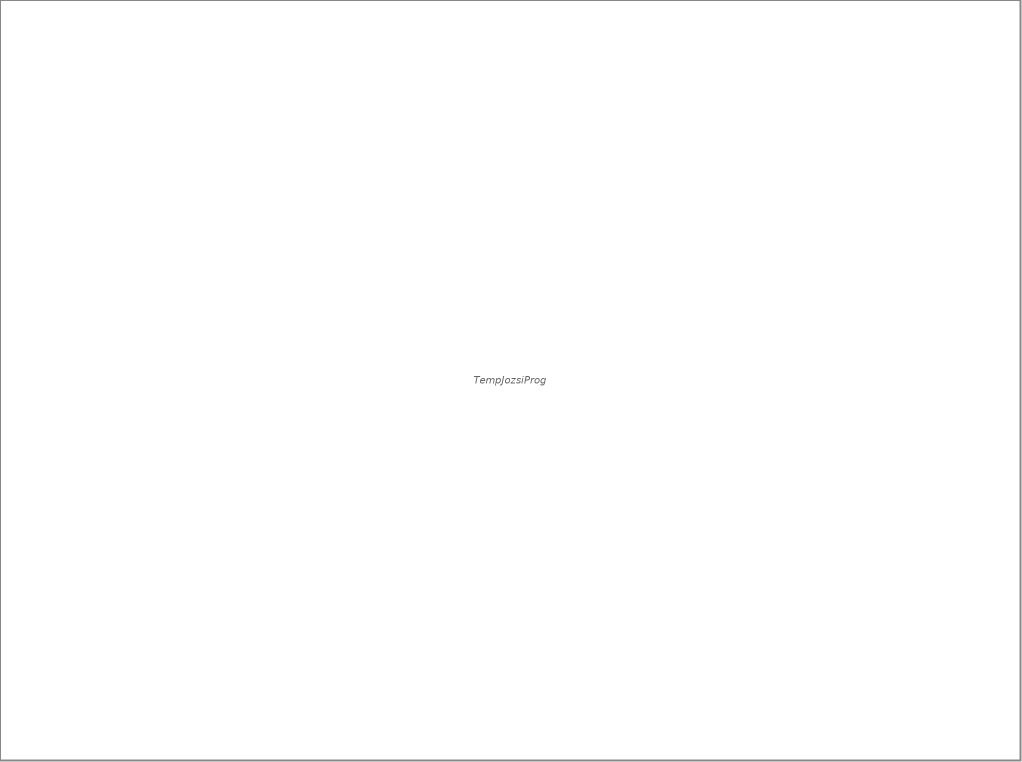
VISUALIZATION TempJozsi  // 1022x762
    TabControl (0,0 1020x760)
        shows TempJozsiProg()
        shows TempJozsiHajlitok()
        shows TempJozsiNTC()
        [0]: TabTitle=Program
END_VISUALIZATION

(* stored: Version 1.1.0.1, ProductVersion 3.1.4024.11
   Visu TempJozsi: Id {b7334e3f-a3ee-4361-8854-2b0bbfc3a799} *)
